FUNCTION_BLOCK FB_Pulse
VAR_INPUT
	bEnable		: BOOL;		//When TRUE, bPulse will be on for tTimeOn and off for tTimeOff
	tTimeOn		: TIME;		//Time bPulse is On
	tTimeOff	: TIME;		//Time bPulse is Off
END_VAR
VAR_OUTPUT
	bPulse		: BOOL;
END_VAR
VAR
	fbTON		: TON;
	fbTOF		: TOF;
END_VAR

(*
//*****************************************************************Notes**********************************************************\\



  
  
//*****************************************************************Revs**********************************************************\\
   (          who            )(    Date    ) (   Rev     ) (								Disc						)
     Chris Mauban			 	2016.05.06		0.00.01		Initial Code
				
     		 								 				
	 						
	
//*****************************************************************Code**********************************************************\\
*)
fbTON(IN:= bEnable AND NOT fbTOF.Q, PT:= tTimeOn, Q=> , ET=> );
fbTOF(IN:= fbTON.Q, PT:= tTimeOff, Q=> , ET=> );

IF bEnable THEN
	bPulse := fbTON.M;
ELSE
	bPulse := FALSE;
END_IF

END_FUNCTION_BLOCK

(* stored: Version 1.1.0.1, ProductVersion 3.1.4022.3
   POU FB_Pulse: Id {b2e8c1b1-02a8-4d75-b9ad-31266dda4a13}, SpecialFunc None *)
